// TIA Portal V16 export
// export: Created 2023-11-14T19:43:11.1722189Z, ExportSetting WithDefaults, DisplayName Totally Integrated Automation Portal, DisplayVersion V16, DisplayName TIA Portal Version Control Interface, DisplayVersion V16, DisplayName TIA Portal Openness, DisplayVersion V16, DisplayName SINAMICS Startdrive Advanced, DisplayVersion V16, DisplayName SINAMICS Startdrive G130, G150, S120, S150, SINAMICS MV, S210, DisplayVersion V16, DisplayName SINAMICS Startdrive G110M, G120, G120C, G120D, G120P, DisplayVersion V16, DisplayName STEP 7 Professional, DisplayVersion V16, DisplayName STEP 7 Safety, DisplayVersion V16, DisplayName WinCC Professional, DisplayVersion V16
ORGANIZATION_BLOCK "Cyclic interrupt"   // OB30, LAD, CyclicInterrupt
{ S7_Optimized_Access := 'TRUE' }
VERSION : 0.1
// stored: AutoNumber true, IsIECCheckEnabled false, SetENOAutomatically false
   VAR_INPUT
      Initial_Call : Bool;   // Initial call of this OB
      Event_Count : Int;   // Events discarded
   END_VAR
BEGIN

REGION Network 1
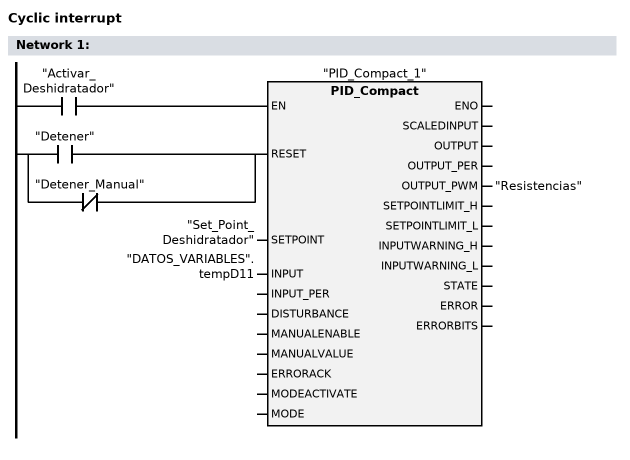
   RUNG wire#powerrail
      Contact( "Activar_Deshidratador" )
      "PID_Compact_1".PID_Compact(Reset := wire#w1, Setpoint := "Set_Point_Deshidratador", Input := "DATOS_VARIABLES".tempD11, Input_PER :=, Disturbance :=, ManualEnable :=, ManualValue :=, ErrorAck :=, ModeActivate :=, Mode :=, ScaledInput =>, Output =>, Output_PER =>, Output_PWM => "Resistencias", SetpointLimit_H =>, SetpointLimit_L =>, InputWarning_H =>, InputWarning_L =>, State =>, Error =>, ErrorBits =>)
   END_RUNG
   RUNG wire#powerrail
      Contact( "Detener" )
   END_RUNG wire#w1
   RUNG wire#powerrail
      I_Contact( "Detener_Manual" )
   END_RUNG wire#w1
   // the same network as SCL:
   IF "Activar_Deshidratador" THEN
       "PID_Compact_1"(Reset := "Detener" OR NOT "Detener_Manual",   // PID_Compact
                       Setpoint := "Set_Point_Deshidratador",
                       Input := "DATOS_VARIABLES".tempD11,
                       Output_PWM => "Resistencias");
   END_IF;
END_REGION
END_ORGANIZATION_BLOCK
